DATA_BLOCK "DB_StarDeltaIO"
{ S7_Optimized_Access := 'TRUE' }
VERSION : 0.1
NON_RETAIN
VAR
    Starter : "UDT_StarDeltaStarterIO";
END_VAR

BEGIN
END_DATA_BLOCK
